TYPE RobotStatusGW1 :
STRUCT
	Status : STRING;
END_STRUCT
END_TYPE

(* stored: Version 1.1.0.1, ProductVersion 3.1.4024.11
   DUT RobotStatusGW1: Id {72821bf8-befc-4067-90b9-0c1ae9f9c536} *)
